(* PLC project TC3_TE1400_GeneratedModule_ModelBase2FM_FB, Beckhoff Automation GmbH & Co. KG TwinCAT 3 Function - TE1400 1.2.1228 *)
(* stored: companyURL www.beckhoff.com, creationDateTime 2017-03-29T12:16:05 *)

TYPE E_TcMatSimDataAreaType : (NotSpecified := 0, Standard, InputSrc, InputDst, OutputSrc, OutputDst, InternalDa, MArea, RetainDa);
END_TYPE

TYPE ST_TcMatSimObjectDataAreaInfo : STRUCT
  pPlcVar : PVOID;
  pModuleProcImg : PVOID;
  nSize : UDINT;
  nDataAreaId : UDINT;
  eDataAreaType : E_TcMatSimDataAreaType;
END_STRUCT;
END_TYPE

{attribute 'pack_mode' := '4'}
TYPE ST_ModelBase2FM_InitData : STRUCT
  Header : TComInitDataHdr;
  CallByHdr : TComInitDataElmHdr;
  CallBy : TctModuleCallByType;
  ExecutionSequenceHdr : TComInitDataElmHdr;
  ExecutionSequence : TctModuleExecutionSequenceType;
  StepSizeHdr : TComInitDataElmHdr;
  StepSize : TctStepSizeType;
  ExtendedFileAccessOIDHdr : TComInitDataElmHdr;
  ExtendedFileAccessOID : OTCID;
  ExtModeParametersHdr : TComInitDataElmHdr;
  ExtModeParameters : TctExtModeParametersType;
  ExecuteModelCodeHdr : TComInitDataElmHdr;
  ExecuteModelCode : BOOL;
  ModelParametersHdr : TComInitDataElmHdr;
  ModelParameters : P_model_base_2fm_T;
  ContextInfoArr_0_TaskOidHdr : TComInitDataElmHdr;
  ContextInfoArr_0_TaskOid : OTCID;
  ContextInfoArr_0_TaskPriorityHdr : TComInitDataElmHdr;
  ContextInfoArr_0_TaskPriority : UDINT;
  ContextInfoArr_0_TaskCycleTimeNsHdr : TComInitDataElmHdr;
  ContextInfoArr_0_TaskCycleTimeNs : UDINT;
  ContextInfoArr_0_TaskPortHdr : TComInitDataElmHdr;
  ContextInfoArr_0_TaskPort : UINT;
  ContextInfoArr_0_TaskSortOrderHdr : TComInitDataElmHdr;
  ContextInfoArr_0_TaskSortOrder : UDINT;
END_STRUCT;
END_TYPE

TYPE ST_ModelBase2FM_Input : STRUCT
  StatusWord_joint1 : UINT;
  MotorEncoder_joint1 : DINT;
  JointAbsEnc_joint1 : DINT;
  MotorCurrentAct_joint1 : INT;
  StatusWord_joint2 : UINT;
  MotorEncoder_joint2 : DINT;
  JointAbsEnc_joint2 : DINT;
  MotorCurrentAct_joint2 : INT;
  FTch1 : REAL;
  FTch2 : REAL;
  FTch3 : REAL;
  FTch4 : REAL;
  FTch5 : REAL;
  FTch6 : REAL;
  StatusWord_joint3 : UINT;
  MotorEncoder_joint3 : DINT;
  JointAbsEnc_joint3 : DINT;
  MotorCurrentAct_joint3 : INT;
  StatusWord_joint4 : UINT;
  MotorEncoder_joint4 : DINT;
  JointAbsEnc_joint4 : DINT;
  MotorCurrentAct_joint4 : INT;
  FTch7 : REAL;
  FTch8 : REAL;
  FTch9 : REAL;
  FTch10 : REAL;
  FTch11 : REAL;
  FTch12 : REAL;
END_STRUCT;
END_TYPE

TYPE ST_ModelBase2FM_Output : STRUCT
  EnableCircuit : BOOL;
  ControlWord_joint1 : UINT;
  ModesOfOperation_joint1 : SINT;
  TargetCurrent_joint1 : INT;
  ControlWord_joint2 : UINT;
  ModesOfOperation_joint2 : SINT;
  TargetCurrent_joint2 : INT;
  pause_logger : BOOL;
  EnableCircuit1 : BOOL;
  ControlWord_joint3 : UINT;
  ModesOfOperation_joint3 : SINT;
  TargetCurrent_joint3 : INT;
  ControlWord_joint4 : UINT;
  ModesOfOperation_joint4 : SINT;
  TargetCurrent_joint4 : INT;
END_STRUCT;
END_TYPE

FUNCTION_BLOCK FB_TcMatSimObject
  VAR_INPUT
    bWriteFbInputValues : BOOL := TRUE;  (* set this flag to write FB input values to the TcComObject's input DataAreas. This will overwrite the mapped input values before module execution. Set to FALSE to read the mapped input values from the TcComObject to the FB. *)
  END_VAR
  VAR
    pDataAreas : POINTER TO ST_TcMatSimObjectDataAreaInfo;  (* process image src and dst pointers and sizes *)
    nDataAreas : UDINT;
    ipObjSrv : ITComObjectServer;  (* global interface pointers *)
    ipTcComObj : ITComObject;  (* object interface pointers *)
    ipTcCyclic : ITcCyclic;
    ipTcPostCyclic : ITcPostCyclic;
    ipTcAdi : ITcADI;
    ipTask : ITcTask;  (* task interface pointers *)
    pInitData : POINTER TO TComInitDataHdr;  (* initial parameters *)
    hResult : HRESULT;  (* hResult of interface calls (0 if no error) *)
    moduleClsId : CLSID;  (* module class ID *)
    assignedClsId : CLSID;  (* expected/desired module class ID *)
    bClassIdVerified : BOOL;
    bDynInstance : BOOL;  (* flag indicating whether the module instance was created dynamically *)
    eInitialObjState : TCOM_STATE := TCOM_STATE.TCOM_STATE_INIT;  (* the object state at the time FB_init was called, FB_exit will try to switch to this state (only if this means to shift down) *)
  END_VAR

            
          

{attribute 'object_name' := 'ReleaseTcComInterface'}
METHOD ReleaseTcComInterface : HRESULT
  VAR
    nStateChangeCnt : DINT := 0;
  END_VAR
                  
IF (ipTcComObj<>0) THEN
  WHILE (State>eInitialObjState AND nStateChangeCnt<1000) DO
    State := eInitialObjState;
    nStateChangeCnt := nStateChangeCnt+1;
  END_WHILE
  ReleaseObjInterfaces();
  IF (bDynInstance) THEN
    ReleaseTcComInterface := TC3_MODULE.FW_ObjMgr_DeleteInstance(ADR(ipTcComObj));
  ELSE
    ipTcComObj.TcRelease();
  END_IF
  ipTcComObj := 0;
END_IF
                  
                
END_METHOD

{attribute 'object_name' := 'ReleaseObjInterfaces'}
METHOD ReleaseObjInterfaces : HRESULT
                  
// release interface pointers
IF (ipTcCyclic<>0) THEN
  ipTcCyclic.TcRelease();
  ipTcCyclic := 0;
END_IF
IF (ipTcPostCyclic<>0) THEN
  ipTcPostCyclic.TcRelease();
  ipTcPostCyclic := 0;
END_IF
IF (ipTcAdi<>0) THEN
  ipTcAdi.TcRelease();
  ipTcAdi := 0;
END_IF
                  
                
END_METHOD

{attribute 'object_name' := 'Internal_SetObjState'}
METHOD Internal_SetObjState
  VAR_INPUT
    hr : REFERENCE TO HRESULT;
    nextState : TCOM_STATE;
  END_VAR
                  
// verify class id
IF (SUCCEEDED(hr)) THEN
  hr := VerifyClassId();
END_IF

// switch object state
IF (SUCCEEDED(hr) AND nextState>=TCOM_STATE_INIT) THEN
  IF (ipTcComObj=0) THEN
    hr := Tc2_System.E_HRESULTAdsErr.NOINTERFACE;
  END_IF
  IF (ipObjSrv=0) THEN
    hr := Tc2_System.E_HRESULTAdsErr.NOINTERFACE;
  END_IF
  IF (SUCCEEDED(hr)) THEN
    hr := ipTcComObj.TcSetObjState(nextState,ipObjSrv,pInitData);
  END_IF
END_IF
                  
                
END_METHOD

{attribute 'object_name' := 'FB_init'}
METHOD FB_init : BOOL
  VAR_INPUT
    bInitRetains : BOOL;  (* init retain variables *)
    bInCopyCode : BOOL;  (* Online Change *)
    oid : OTCID;
  END_VAR
                  
FB_init := SUCCEEDED(Init(oid));
                  
                
END_METHOD

{attribute 'object_name' := 'GetObjPara'}
METHOD GetObjPara : HRESULT
  VAR_INPUT
    pid : PTCID;
    nData : UDINT;
    pData : PVOID;
  END_VAR
                  
IF (ipTcComObj=0) THEN
  GetObjPara := Tc2_System.E_HRESULTAdsErr.NOINTERFACE;
END_IF

IF (SUCCEEDED(GetObjPara)) THEN
  GetObjPara := ipTcComObj.TcGetObjPara(pid:=pid,nData,pData,0);
END_IF
                  
                
END_METHOD

{attribute 'object_name' := 'QueryObjInterface'}
METHOD QueryObjInterface
  VAR_INPUT
    hr : REFERENCE TO HRESULT;
    iid : REFERENCE TO IID;
    pipItf : POINTER TO ITcUnknown;
  END_VAR
  VAR CONSTANT
    pNull : PVOID := 0;
  END_VAR
                  
IF (SUCCEEDED(hr)) THEN
  IF (ipTcComObj=0) THEN
    hr := Tc2_System.E_HRESULTAdsErr.NOINTERFACE;
  ELSIF (pipItf^=ULINT_TO_DWORD(pNull)) THEN
    hr := ipTcComObj.TcQueryInterface(iid:= iid, pipItf:=pipItf);
  END_IF
END_IF
                  
                
END_METHOD

{attribute 'object_name' := 'SaveOnlineParametersForInit'}
METHOD SaveOnlineParametersForInit : HRESULT
  VAR
    idx : UINT;
    pInitElemHdr : POINTER TO TComInitDataElmHdr;
    pData : PVOID;
    nData : UDINT;
  END_VAR
  VAR CONSTANT
    nInitDataAlignment : UDINT := 4;
  END_VAR
                  IF (pInitData<>0) THEN
  pInitElemHdr := pInitData + SIZEOF(pInitData^);
  FOR idx:=1 TO pInitData^.uiElmCnt DO
    pData := pInitElemHdr + ULINT_TO_DWORD(SIZEOF(pInitElemHdr^));
    nData := pInitElemHdr^.cbData;
    SaveOnlineParametersForInit := GetObjPara(pInitElemHdr^.indexOffset,nData,pData);
    IF (FAILED(SaveOnlineParametersForInit)) THEN
      RETURN;
    END_IF
    pInitElemHdr := pData + (nInitDataAlignment*((nData + nInitDataAlignment - 1)/nInitDataAlignment));
  END_FOR
ELSE
	SaveOnlineParametersForInit := Tc2_System.E_HRESULTAdsErr.NOTINIT;
END_IF
                  
                
END_METHOD

{attribute 'object_name' := 'ResetHresult'}
METHOD ResetHresult
                  hResult := S_OK;
                
END_METHOD

{attribute 'object_name' := 'Execute'}
METHOD Execute : HRESULT
  VAR
    nDaIdx : UDINT;
    pCurDataArea : POINTER TO ST_TcMatSimObjectDataAreaInfo;
  END_VAR
                  
IF (SUCCEEDED(hResult)) THEN
  hResult := VerifyClassId();
END_IF

IF (SUCCEEDED(hResult) AND State<>TCOM_STATE_OP) THEN
  hResult := Tc2_System.E_HRESULTAdsErr.NOTREADY;
END_IF

// get image pointers
IF (SUCCEEDED(hResult)) THEN
  GetImagePtrs(hResult);
END_IF

// copy inputs
IF (pDataAreas<>0 AND bWriteFbInputValues) THEN
  FOR nDaIdx:=0 TO nDataAreas-1 DO
    IF (FAILED(hResult))THEN
      CONTINUE;
    END_IF
    pCurDataArea := pDataAreas + nDaIdx*SIZEOF(ST_TcMatSimObjectDataAreaInfo);
    IF ((pCurDataArea^.eDataAreaType <> E_TcMatSimDataAreaType.InputDst))THEN
      CONTINUE;
    END_IF
    IF (pCurDataArea^.pModuleProcImg<>0 AND pCurDataArea^.pPlcVar<>0) THEN
      MEMCPY(pCurDataArea^.pModuleProcImg,pCurDataArea^.pPlcVar,pCurDataArea^.nSize);
    ELSE
      hResult := Tc2_System.E_HRESULTAdsErr.NOINTERFACE;
    END_IF
  END_FOR
END_IF

// call cycle update
IF (SUCCEEDED(hResult)) THEN
  IF (ipTcCyclic<>0) THEN
    hResult := ipTcCyclic.CycleUpdate(ipTask:= ipTask, ipCaller:= 0, context:= 0);
  ELSE
    hResult := Tc2_System.E_HRESULTAdsErr.NOINTERFACE;
  END_IF
END_IF

// copy outputs
IF (pDataAreas<>0) THEN
  FOR nDaIdx:=0 TO nDataAreas-1 DO
    IF (FAILED(hResult))THEN
      CONTINUE;
    END_IF
    pCurDataArea := pDataAreas + nDaIdx*SIZEOF(ST_TcMatSimObjectDataAreaInfo);
    IF ((pCurDataArea^.eDataAreaType = E_TcMatSimDataAreaType.OutputSrc) OR NOT bWriteFbInputValues) THEN
      IF (pCurDataArea^.pModuleProcImg<>0 AND pCurDataArea^.pPlcVar<>0) THEN
        MEMCPY(pCurDataArea^.pPlcVar,pCurDataArea^.pModuleProcImg,pCurDataArea^.nSize);
      ELSE
        hResult := Tc2_System.E_HRESULTAdsErr.NOINTERFACE;
      END_IF
    END_IF
  END_FOR
END_IF


// call post cyclic update
IF (SUCCEEDED(hResult)) THEN
  IF (ipTcPostCyclic<>0) THEN
    hResult := ipTcPostCyclic.PostCyclicUpdate(ipTask:= 0, ipCaller:= 0, context:= 0);
  ELSE
    hResult := Tc2_System.E_HRESULTAdsErr.NOINTERFACE;
  END_IF
END_IF

ReleaseImagePtrs();

Execute := hResult;
                  
                
END_METHOD

{attribute 'object_name' := 'GetImagePtrs'}
METHOD GetImagePtrs
  VAR_INPUT
    hr : REFERENCE TO HRESULT;
  END_VAR
  VAR
    nDaIdx : UDINT;
    pCurDataArea : POINTER TO ST_TcMatSimObjectDataAreaInfo;
  END_VAR
                  
IF (ipTcAdi=0) THEN
  hr := Tc2_System.E_HRESULTAdsErr.NOINTERFACE;
END_IF
IF(State<>TCOM_STATE_OP)THEN
  hr := Tc2_System.E_HRESULTAdsErr.INVALIDSTATE;
END_IF


// get pointers to process images
IF (pDataAreas<>0) THEN
  FOR nDaIdx:=0 TO nDataAreas-1 DO
    pCurDataArea := pDataAreas + nDaIdx*SIZEOF(ST_TcMatSimObjectDataAreaInfo);
    IF (FAILED(hr))THEN
      CONTINUE;
    END_IF
    IF ((pCurDataArea^.eDataAreaType <> E_TcMatSimDataAreaType.InputDst) AND (pCurDataArea^.eDataAreaType <> E_TcMatSimDataAreaType.OutputSrc))THEN
      CONTINUE;
    END_IF
    IF (pCurDataArea^.pModuleProcImg=0 AND pCurDataArea^.nSize>0) THEN
      hr := ipTcAdi.GetImagePtr(size:= pCurDataArea^.nSize , offs:=0 , adi_x:=pCurDataArea^.nDataAreaId , ppData:=ADR(pCurDataArea^.pModuleProcImg));
    END_IF
  END_FOR
END_IF

IF (FAILED(hr)) THEN
  ReleaseImagePtrs();
END_IF
                  
                
END_METHOD

{attribute 'object_name' := 'VerifyClassId'}
METHOD VerifyClassId : HRESULT
  VAR
    emptyClsId : CLSID;
  END_VAR
                  memset(ADR(emptyClsId),0,SIZEOF(emptyClsId));
IF (bClassIdVerified) THEN
  // class ID was already verified
  VerifyClassId := Tc2_System.E_HRESULTAdsErr.HRESULT_ADS_NOERROR;
ELSIF (memcmp(ADR(assignedClsId),ADR(emptyClsId),SIZEOF(assignedClsId))=0) THEN
  // skip class ID verification if no assignedClsId specified
  VerifyClassId := Tc2_System.E_HRESULTAdsErr.HRESULT_ADS_NOERROR;
ELSE
  // verify class ID
  VerifyClassId := ReadModuleClassId();

  IF (SUCCEEDED(VerifyClassId)) THEN
    IF (memcmp(ADR(assignedClsId),ADR(moduleClsId),SIZEOF(assignedClsId))<>0) THEN
     VerifyClassId := Tc2_System.E_HRESULTAdsErr.INVALIDCLSID;
    END_IF
  END_IF
  bClassIdVerified := SUCCEEDED(VerifyClassId);
END_IF
                  
                
END_METHOD

{attribute 'object_name' := 'SetObjPara'}
METHOD SetObjPara : HRESULT
  VAR_INPUT
    pid : PTCID;
    nData : UDINT;
    pData : PVOID;
  END_VAR
                  
IF (ipTcComObj=0) THEN
  SetObjPara := Tc2_System.E_HRESULTAdsErr.NOINTERFACE;
END_IF

IF (SUCCEEDED(SetObjPara)) THEN
  SetObjPara := ipTcComObj.TcSetObjPara(pid:=pid,nData,pData,0);
END_IF
                  
                
END_METHOD

{attribute 'object_name' := 'QueryTcComInterface'}
METHOD QueryTcComInterface
  VAR_INPUT
    hr : REFERENCE TO HRESULT;
    oid : OTCID;
  END_VAR
                  
IF (ipObjSrv=0) THEN
  hr := Tc2_System.E_HRESULTAdsErr.NOINTERFACE;
END_IF

IF (SUCCEEDED(hr) AND ipTcComObj=0) THEN
  bDynInstance := FALSE;
  IF(oid>0) THEN
    // query interface of existing object
    hr := ipObjSrv.TcQueryObjectInterface(oid,IID_ITComObject,ADR(ipTcComObj));
  ELSE
    // create new instance and get the object interface
    hr := ipObjSrv.TcCreateInstance(assignedClsId,IID_ITComObject,ADR(ipTcComObj));
    IF (SUCCEEDED(hr)) THEN
      bDynInstance := TRUE;
      hr := ipTcComObj.TcSetObjectId(OTCID_CreateNewId);
    END_IF
  END_IF
  IF (SUCCEEDED(hr)) THEN
    eInitialObjState := State;
  END_IF
END_IF
                  
                
END_METHOD

{attribute 'object_name' := 'ReleaseImagePtrs'}
METHOD ReleaseImagePtrs : HRESULT
  VAR
    nDaIdx : UDINT;
    pCurDataArea : POINTER TO ST_TcMatSimObjectDataAreaInfo;
  END_VAR
                  
IF (ipTcAdi=0) THEN
  ReleaseImagePtrs := Tc2_System.E_HRESULTAdsErr.NOINTERFACE;
END_IF

IF (SUCCEEDED(ReleaseImagePtrs) AND pDataAreas<>0) THEN
  // release pointers to the simulink module process images
  FOR nDaIdx:=0 TO nDataAreas-1 DO
    pCurDataArea := pDataAreas + nDaIdx*SIZEOF(ST_TcMatSimObjectDataAreaInfo);

    IF (pCurDataArea^.pModuleProcImg<>0) THEN
      ipTcAdi.ReleaseImagePtr(pData:=pCurDataArea^.pModuleProcImg);
      pCurDataArea^.pModuleProcImg := 0;
    END_IF
  END_FOR
END_IF
                  
                
END_METHOD

{attribute 'object_name' := 'FB_exit'}
METHOD FB_exit : BOOL
  VAR_INPUT
    bInCopyCode : BOOL;  (* Online Change *)
  END_VAR
                  
IF (NOT bInCopyCode) THEN
  IF (ipObjSrv<>0) THEN
    ipObjSrv.TcRelease();
    ipObjSrv := 0;
  END_IF

  ReleaseTcComInterface();
END_IF
                  
                
END_METHOD

{attribute 'object_name' := 'InitObjName'}
METHOD InitObjName
  VAR_INPUT
    hr : REFERENCE TO HRESULT;
  END_VAR
  VAR
    objectName : STRING(255) := 'TempContr_PlcRtFbInstance';
    oid : OTCID;
  END_VAR
                  
IF (SUCCEEDED(hr)) THEN
  hr := ipTcComObj.TcGetObjectId(oid);
END_IF

IF (SUCCEEDED(hr) and bDynInstance) THEN
  objectName := TC2_STANDARD.CONCAT(objectName,'_');
  objectName := TC2_STANDARD.CONCAT(objectName,UDINT_TO_STRING(oid));
  hr := ipTcComObj.TcSetObjectName(ADR(objectName));
END_IF
                  
                
END_METHOD

{attribute 'object_name' := 'SetObjState'}
METHOD SetObjState : HRESULT
  VAR_INPUT
    finalState : TCOM_STATE;
  END_VAR
  VAR
    bShiftUp : BOOL;
    bShiftDown : BOOL;
    currentState : TCOM_STATE;
  END_VAR
                  
currentState := State;

bShiftUp := finalState>currentState;
bShiftDown := finalState<currentState;

// do not switch up on error
IF (FAILED(hresult)) THEN
  bShiftUp := FALSE;
END_IF
// reset existing error on switching down
IF (bShiftDown) THEN
  ResetHresult();
END_IF

// prepared state switch
CASE currentState OF
  TCOM_STATE_INIT:
    IF(bShiftUp) THEN
      QueryTcComInterface(hResult,0);
      Internal_SetObjState(hResult,TCOM_STATE.TCOM_STATE_PREOP);
      InitObjName(hResult);
    END_IF

  TCOM_STATE_PREOP:
    IF(bShiftUp) THEN
      Internal_SetObjState(hResult,TCOM_STATE.TCOM_STATE_SAFEOP);
      QueryObjInterfaces(hResult);
    ELSIF (bShiftDown) THEN
      Internal_SetObjState(hResult,TCOM_STATE.TCOM_STATE_INIT);
    END_IF

  TCOM_STATE_SAFEOP:
    IF(bShiftUp) THEN
      Internal_SetObjState(hResult,TCOM_STATE.TCOM_STATE_OP);
      QueryObjInterfaces(hResult);
    ELSIF (bShiftDown) THEN
      Internal_SetObjState(hResult,TCOM_STATE.TCOM_STATE_PREOP);
      ReleaseObjInterfaces();
    END_IF


  TCOM_STATE_OP:
    IF (bShiftDown) THEN
      Internal_SetObjState(hResult,TCOM_STATE.TCOM_STATE_SAFEOP);
    END_IF
END_CASE

SetObjState := hResult;
                  
                
END_METHOD

{attribute 'object_name' := 'QueryObjInterfaces'}
METHOD QueryObjInterfaces
  VAR_INPUT
    hr : REFERENCE TO HRESULT;
  END_VAR
                  
IF(State<TCOM_STATE_PREOP)THEN
  hr := Tc2_System.E_HRESULTAdsErr.INVALIDSTATE;
END_IF

//cyclic interface
QueryObjInterface(hr,IID_ITCCYCLIC,ADR(ipTcCyclic));
//post cyclic interface
QueryObjInterface(hr,IID_ITCPOSTCYCLIC,ADR(ipTcPostCyclic));
//adi interface
QueryObjInterface(hr,IID_ITcADI,ADR(ipTcAdi));
                  
                
END_METHOD

{attribute 'object_name' := 'Init'}
METHOD Init : HRESULT
  VAR_INPUT
    oid : OTCID;
  END_VAR
                  
// preinitialize variables
memset(ADR(moduleClsId),0,SIZEOF(moduleClsId));
bClassIdVerified := FALSE;
hResult := Tc2_System.E_HRESULTAdsErr.HRESULT_ADS_NOERROR;

// get object server
IF (ipObjSrv=0) THEN
  hResult := FW_ObjMgr_GetObjectServer(_AppInfo.ObjId,ADR(ipObjSrv));
END_IF

// try to get object interfaces
IF (SUCCEEDED(hresult)) THEN
  QueryTcComInterface(hResult,oid);
END_IF

// verify class id
IF (SUCCEEDED(hresult)) THEN
  hresult := VerifyClassId();
END_IF

// query interfaces, if the current state is higher than INIT
IF (SUCCEEDED(hresult) AND State>TCOM_STATE.TCOM_STATE_INIT) THEN
  QueryObjInterfaces(hResult);
END_IF

// return value
Init := hresult;
                  
                
END_METHOD

{attribute 'object_name' := 'ReadModuleClassId'}
METHOD ReadModuleClassId : HRESULT
  VAR
    emptyClsId : CLSID;
  END_VAR
                  memset(ADR(emptyClsId),0,SIZEOF(emptyClsId));
IF (memcmp(ADR(moduleClsId),ADR(emptyClsId),SIZEOF(moduleClsId))=0) THEN
  IF (ipTcComObj=0) THEN
    ReadModuleClassId := Tc2_System.E_HRESULTAdsErr.NOINTERFACE;
  END_IF

  //objectClsId := clsid;
  IF (SUCCEEDED(ReadModuleClassId)) THEN
    ReadModuleClassId := ipTcComObj.GetClassId(moduleClsId);
  END_IF
END_IF
                
END_METHOD

METHOD PUBLIC AssignClassId
VAR_INPUT
	clsId : CLSID;
END_VAR
                  assignedClsId := clsId;
bClassIdVerified := false;
                  
                
END_METHOD

PROPERTY Error : BOOL
GET
                    Error := FAILED(hResult);
                  
END_GET
END_PROPERTY

METHOD PUBLIC SetDataAreaInfo
VAR_INPUT
  pDataAreas: POINTER TO ST_TcMatSimObjectDataAreaInfo;
  nDataAreas: UDINT;
END_VAR
                  
THIS^.nDataAreas := nDataAreas;
THIS^.pDataAreas := pDataAreas;
                  
                
END_METHOD

METHOD PUBLIC SetInitDataInfo
VAR_INPUT
  pInitData : POINTER TO TComInitDataHdr;
END_VAR
                  this^.pInitData := pInitData;
                
END_METHOD

PROPERTY ClassId : CLSID
GET
                    hResult := ReadModuleClassId();
ClassId := moduleClsId;
                    
                  
END_GET
END_PROPERTY

PROPERTY State : TCOM_STATE
GET
  VAR
    hr : HRESULT := S_OK;
    eObjState : TCOM_STATE;
  END_VAR
                    
IF (ipTcComObj<>0) THEN
  hr := ipTcComObj.TcGetObjState(ADR(eObjState));
IF (FAILED(hr)) THEN
  eObjState := TCOM_STATE.TCOM_STATE_INIT;
END_IF
ELSE
  eObjState := TCOM_STATE.TCOM_STATE_INIT;
END_IF
State := eObjState;
                    
                  
END_GET
SET
                    SetObjState(State);
                  
END_SET
END_PROPERTY

PROPERTY ErrorCode : HRESULT
GET
                    ErrorCode := hResult;
                  
END_GET
END_PROPERTY
END_FUNCTION_BLOCK

{attribute 'TcDependOnClassFactory' := 'ModelBase2FM'}
FUNCTION_BLOCK FB_ModelBase2FM EXTENDS FB_TcMatSimObject
  VAR_INPUT
    stInput : ST_ModelBase2FM_Input;
  END_VAR
  VAR_OUTPUT
    stOutput : ST_ModelBase2FM_Output;
  END_VAR
  VAR
    stInitData : ST_ModelBase2FM_InitData;
    arrDataAreas : ARRAY[1..2] OF ST_TcMatSimObjectDataAreaInfo;
    bParametersVerified : BOOL;
  END_VAR

            
          

{attribute 'object_name' := 'Internal_SetObjState'}
METHOD Internal_SetObjState
  VAR_INPUT
    hr : REFERENCE TO HRESULT;
    nextState : TCOM_STATE;
  END_VAR
                  
// update pointer to InitData structure
SetInitDataInfo(ADR(stInitData));
// call base method
SUPER^.Internal_SetObjState(hr,nextState);
                  
                
END_METHOD

{attribute 'object_name' := 'SaveOnlineParametersForInit'}
METHOD SaveOnlineParametersForInit : HRESULT
  VAR
    idx : UINT;
    pInitElemHdr : POINTER TO TComInitDataElmHdr;
    pData : PVOID;
    nData : UDINT;
  END_VAR
  VAR CONSTANT
    nInitDataAlignment : UDINT := 4;
  END_VAR
                  
// update pointer to InitData structure
SetInitDataInfo(ADR(stInitData));
// call base method
SaveOnlineParametersForInit := SUPER^.SaveOnlineParametersForInit();
                  
                
END_METHOD

METHOD FB_init : BOOL
  VAR_INPUT
    bInitRetains : BOOL;  (* if TRUE, the retain variables are initialized (warm start / cold start) *)
    bInCopyCode : BOOL;  (* if TRUE, the instance afterwards gets moved into the copy code (online change) *)
    oid : OTCID;
  END_VAR
  VAR
    clsId : CLSID;
  END_VAR
                  
// initialize flags
bParametersVerified := false;
                    
// set module class id for compatibility check
clsId.Data1 := 16#36160af7;
clsId.Data2 := 16#e4ae;
clsId.Data3 := 16#44ca;
clsId.Data4[0] := 16#81;
clsId.Data4[1] := 16#8b;
clsId.Data4[2] := 16#1e;
clsId.Data4[3] := 16#af;
clsId.Data4[4] := 16#06;
clsId.Data4[5] := 16#99;
clsId.Data4[6] := 16#96;
clsId.Data4[7] := 16#6e;

AssignClassId(clsId);
                    
// initialize InitData structure with default values              
stInitData.CallByHdr.indexGroup := 0;
stInitData.CallByHdr.indexOffset := 16#00000000;
stInitData.CallByHdr.cbData := SIZEOF(stInitData.CallBy);
stInitData.CallBy := TctModuleCallByType.CyclicTask;
stInitData.ExecutionSequenceHdr.indexGroup := 0;
stInitData.ExecutionSequenceHdr.indexOffset := 16#00000001;
stInitData.ExecutionSequenceHdr.cbData := SIZEOF(stInitData.ExecutionSequence);
stInitData.ExecutionSequence := TctModuleExecutionSequenceType.StateUpdateAfterOutputMapping;
stInitData.StepSizeHdr.indexGroup := 0;
stInitData.StepSizeHdr.indexOffset := 16#00000002;
stInitData.StepSizeHdr.cbData := SIZEOF(stInitData.StepSize);
stInitData.StepSize := TctStepSizeType.RequireMatchingTaskCycleTime;
stInitData.ExtendedFileAccessOIDHdr.indexGroup := 0;
stInitData.ExtendedFileAccessOIDHdr.indexOffset := 16#00000005;
stInitData.ExtendedFileAccessOIDHdr.cbData := SIZEOF(stInitData.ExtendedFileAccessOID);
stInitData.ExtendedFileAccessOID := 0;
stInitData.ExtModeParametersHdr.indexGroup := 0;
stInitData.ExtModeParametersHdr.indexOffset := 16#bf002000;
stInitData.ExtModeParametersHdr.cbData := SIZEOF(stInitData.ExtModeParameters);
stInitData.ExtModeParameters.ConnectionTimeout := 3;
stInitData.ExtModeParameters.InitIncomingPktBufferSize := 10000;
stInitData.ExtModeParameters.InitOutgoingPktBufferSize := 10000;
stInitData.ExtModeParameters.Activated := 1;
stInitData.ExtModeParameters.AllowExecutionCommands := 1;
stInitData.ExtModeParameters.WaitForStartCommand := 0;
stInitData.ExtModeParameters.AllowParameterChange := 1;
stInitData.ExecuteModelCodeHdr.indexGroup := 0;
stInitData.ExecuteModelCodeHdr.indexOffset := 16#00000008;
stInitData.ExecuteModelCodeHdr.cbData := SIZEOF(stInitData.ExecuteModelCode);
stInitData.ExecuteModelCode := 1;
stInitData.ModelParametersHdr.indexGroup := 0;
stInitData.ModelParametersHdr.indexOffset := 16#83000000;
stInitData.ModelParametersHdr.cbData := SIZEOF(stInitData.ModelParameters);
stInitData.ModelParameters.FM1.HomeLocationOpSpace[0] := 0;
stInitData.ModelParameters.FM1.HomeLocationOpSpace[1] := 0.25;
stInitData.ModelParameters.FM1.HomeLocationSize := 0.01;
stInitData.ModelParameters.FM1.DynModParams[0] := 0.001597109;
stInitData.ModelParameters.FM1.DynModParams[1] := 0.001580786;
stInitData.ModelParameters.FM1.DynModParams[2] := 0.0702826;
stInitData.ModelParameters.FM1.DynModParams[3] := 0.07988736;
stInitData.ModelParameters.FM1.DynModParams[4] := -0;
stInitData.ModelParameters.FM1.DynModParams[5] := 0.1006366;
stInitData.ModelParameters.FM1.DynModParams[6] := -0;
stInitData.ModelParameters.FM1.Actuator1.JointAbsoluteEncoderCounts_rev := 65536;
stInitData.ModelParameters.FM1.Actuator1.AbsEncoderOffset := 5.303223547422882;
stInitData.ModelParameters.FM1.Actuator1.MotorEncoderCounts_rev := 4096;
stInitData.ModelParameters.FM1.Actuator1.FOAWNoiseLevel := 0.0003834951969714103;
stInitData.ModelParameters.FM1.Actuator1.transmissionRatio := 7.2976;
stInitData.ModelParameters.FM1.Actuator1.motorTorqueConstant := 0.08486;
stInitData.ModelParameters.FM1.Actuator1.drivePeakCurrent := 20;
stInitData.ModelParameters.FM1.Actuator1.AbsoluteMaximumTorque_Nm := 8;
stInitData.ModelParameters.FM1.Actuator1.TransmissionSlipAngleGuardMax := 0.08726646259971647;
stInitData.ModelParameters.FM1.Actuator1.JointPositionGuardMin := -0.4363323129985824;
stInitData.ModelParameters.FM1.Actuator1.JointPositionGuardMax := 2.356194490192345;
stInitData.ModelParameters.FM1.Actuator2.JointAbsoluteEncoderCounts_rev := 65536;
stInitData.ModelParameters.FM1.Actuator2.AbsEncoderOffset := 7.340133727728301;
stInitData.ModelParameters.FM1.Actuator2.MotorEncoderCounts_rev := 4096;
stInitData.ModelParameters.FM1.Actuator2.FOAWNoiseLevel := 0.0003834951969714103;
stInitData.ModelParameters.FM1.Actuator2.transmissionRatio := 7.331;
stInitData.ModelParameters.FM1.Actuator2.motorTorqueConstant := 0.08486;
stInitData.ModelParameters.FM1.Actuator2.drivePeakCurrent := 20;
stInitData.ModelParameters.FM1.Actuator2.AbsoluteMaximumTorque_Nm := 8;
stInitData.ModelParameters.FM1.Actuator2.TransmissionSlipAngleGuardMax := 0.08726646259971647;
stInitData.ModelParameters.FM1.Actuator2.JointPositionGuardMin := 0.7853981633974483;
stInitData.ModelParameters.FM1.Actuator2.JointPositionGuardMax := 3.577924966588375;
stInitData.ModelParameters.FM1.FTSensor.MaxAllowableForcesTorqueSensor[0] := 70;
stInitData.ModelParameters.FM1.FTSensor.MaxAllowableForcesTorqueSensor[1] := 70;
stInitData.ModelParameters.FM1.FTSensor.MaxAllowableForcesTorqueSensor[2] := 140;
stInitData.ModelParameters.FM1.FTSensor.MaxAllowableForcesTorqueSensor[3] := 1.4;
stInitData.ModelParameters.FM1.FTSensor.MaxAllowableForcesTorqueSensor[4] := 1.4;
stInitData.ModelParameters.FM1.FTSensor.MaxAllowableForcesTorqueSensor[5] := 1.4;
stInitData.ModelParameters.FM1.FTSensor.TransformationMatrixSide := 1;
stInitData.ModelParameters.FM2.HomeLocationOpSpace[0] := 0;
stInitData.ModelParameters.FM2.HomeLocationOpSpace[1] := 0.25;
stInitData.ModelParameters.FM2.HomeLocationSize := 0.01;
stInitData.ModelParameters.FM2.DynModParams[0] := 0.001597109;
stInitData.ModelParameters.FM2.DynModParams[1] := 0.001580786;
stInitData.ModelParameters.FM2.DynModParams[2] := 0.0702826;
stInitData.ModelParameters.FM2.DynModParams[3] := 0.07988736;
stInitData.ModelParameters.FM2.DynModParams[4] := -0;
stInitData.ModelParameters.FM2.DynModParams[5] := 0.1006366;
stInitData.ModelParameters.FM2.DynModParams[6] := -0;
stInitData.ModelParameters.FM2.Actuator1.JointAbsoluteEncoderCounts_rev := 65536;
stInitData.ModelParameters.FM2.Actuator1.AbsEncoderOffset := 3.23580094055001;
stInitData.ModelParameters.FM2.Actuator1.MotorEncoderCounts_rev := 4096;
stInitData.ModelParameters.FM2.Actuator1.FOAWNoiseLevel := 0.0003834951969714103;
stInitData.ModelParameters.FM2.Actuator1.transmissionRatio := 7.3607;
stInitData.ModelParameters.FM2.Actuator1.motorTorqueConstant := 0.08486;
stInitData.ModelParameters.FM2.Actuator1.drivePeakCurrent := 20;
stInitData.ModelParameters.FM2.Actuator1.AbsoluteMaximumTorque_Nm := 8;
stInitData.ModelParameters.FM2.Actuator1.TransmissionSlipAngleGuardMax := 0.08726646259971647;
stInitData.ModelParameters.FM2.Actuator1.JointPositionGuardMin := -0.4363323129985824;
stInitData.ModelParameters.FM2.Actuator1.JointPositionGuardMax := 2.356194490192345;
stInitData.ModelParameters.FM2.Actuator2.JointAbsoluteEncoderCounts_rev := 65536;
stInitData.ModelParameters.FM2.Actuator2.AbsEncoderOffset := 4.445224359590367;
stInitData.ModelParameters.FM2.Actuator2.MotorEncoderCounts_rev := 4096;
stInitData.ModelParameters.FM2.Actuator2.FOAWNoiseLevel := 0.0003834951969714103;
stInitData.ModelParameters.FM2.Actuator2.transmissionRatio := 7.32214;
stInitData.ModelParameters.FM2.Actuator2.motorTorqueConstant := 0.08486;
stInitData.ModelParameters.FM2.Actuator2.drivePeakCurrent := 20;
stInitData.ModelParameters.FM2.Actuator2.AbsoluteMaximumTorque_Nm := 8;
stInitData.ModelParameters.FM2.Actuator2.TransmissionSlipAngleGuardMax := 0.08726646259971647;
stInitData.ModelParameters.FM2.Actuator2.JointPositionGuardMin := 0.7853981633974483;
stInitData.ModelParameters.FM2.Actuator2.JointPositionGuardMax := 3.577924966588375;
stInitData.ModelParameters.FM2.FTSensor.MaxAllowableForcesTorqueSensor[0] := 70;
stInitData.ModelParameters.FM2.FTSensor.MaxAllowableForcesTorqueSensor[1] := 70;
stInitData.ModelParameters.FM2.FTSensor.MaxAllowableForcesTorqueSensor[2] := 140;
stInitData.ModelParameters.FM2.FTSensor.MaxAllowableForcesTorqueSensor[3] := 1.4;
stInitData.ModelParameters.FM2.FTSensor.MaxAllowableForcesTorqueSensor[4] := 1.4;
stInitData.ModelParameters.FM2.FTSensor.MaxAllowableForcesTorqueSensor[5] := 1.4;
stInitData.ModelParameters.FM2.FTSensor.TransformationMatrixSide := 1;
stInitData.ModelParameters.Lb := 0.07000000000000001;
stInitData.ModelParameters.Lf := 0.238;
stInitData.ModelParameters.Lu := 0.153;
stInitData.ModelParameters.sampleTime := 0.001;
stInitData.ModelParameters.DiscreteDerivative_ICPrevScaled := 0;
stInitData.ModelParameters.DiscreteDerivative_ICPrevScal_b := 0;
stInitData.ModelParameters.DiscreteDerivative_ICPrevScal_a := 0;
stInitData.ModelParameters.DiscreteDerivative_ICPrevScal_h := 0;
stInitData.ModelParameters.DiscreteDerivative_ICPrevScal_j := 0;
stInitData.ModelParameters.DiscreteDerivative_ICPrevScal_k := 0;
stInitData.ModelParameters.DiscreteDerivative_ICPrevScal_i := 0;
stInitData.ModelParameters.DiscreteDerivative_ICPrevScal_o := 0;
stInitData.ModelParameters.CompareToConstant_const := 201;
stInitData.ModelParameters.CompareToConstant_const_b := 0;
stInitData.ModelParameters.CompareToConstant_const_a := 201;
stInitData.ModelParameters.CompareToConstant_const_e := 0;
stInitData.ModelParameters.CompareToConstant_const_aw := 4;
stInitData.ModelParameters.CompareToConstant_const_c := 4;
stInitData.ModelParameters.CompareToConstant1_const := 2.75;
stInitData.ModelParameters.CompareToConstant_const_d := 4;
stInitData.ModelParameters.CompareToConstant_const_m := 4;
stInitData.ModelParameters.CompareToConstant1_const_m := 2.75;
stInitData.ModelParameters.DetectChange_vinit := 0;
stInitData.ModelParameters.DetectChange_vinit_h := 0;
stInitData.ModelParameters.DetectChange_vinit_g := 0;
stInitData.ModelParameters.DetectChange_vinit_b := 0;
stInitData.ModelParameters.ErrorHasOccurred_initial_condit := 0;
stInitData.ModelParameters.ErrorHasOccurred_initial_cond_a := 0;
stInitData.ModelParameters.ErrorHasOccurred_initial_cond_f := 0;
stInitData.ModelParameters.ErrorHasOccurred_initial_cond_k := 0;
stInitData.ModelParameters.DetectRisePositive_vinit := 0;
stInitData.ModelParameters.DetectRisePositive1_vinit := 0;
stInitData.ModelParameters.DetectRisePositive_vinit_c := 0;
stInitData.ModelParameters.DetectRisePositive1_vinit_i := 0;
stInitData.ModelParameters.DetectRisePositive_vinit_m := 0;
stInitData.ModelParameters.DetectRisePositive1_vinit_b := 0;
stInitData.ModelParameters.DetectRisePositive_vinit_n := 0;
stInitData.ModelParameters.DetectRisePositive1_vinit_j := 0;
stInitData.ModelParameters.DetectIncrease_vinit := 0;
stInitData.ModelParameters.DetectIncrease_vinit_f := 0;
stInitData.ModelParameters.JointTorqueDes_Nm_Y0[0] := 0;
stInitData.ModelParameters.JointTorqueDes_Nm_Y0[1] := 0;
stInitData.ModelParameters.Constant3_Value[0] := 0;
stInitData.ModelParameters.Constant3_Value[1] := 0;
stInitData.ModelParameters.JointTorqueDes_Nm_Y0_p[0] := 0;
stInitData.ModelParameters.JointTorqueDes_Nm_Y0_p[1] := 0;
stInitData.ModelParameters.Constant3_Value_h[0] := 0;
stInitData.ModelParameters.Constant3_Value_h[1] := 0;
stInitData.ModelParameters.JointTorqueDes_Nm_Y0_i[0] := 0;
stInitData.ModelParameters.JointTorqueDes_Nm_Y0_i[1] := 0;
stInitData.ModelParameters.Constant3_Value_h5[0] := 0;
stInitData.ModelParameters.Constant3_Value_h5[1] := 0;
stInitData.ModelParameters.JointTorqueDes_Nm_Y0_m[0] := 0;
stInitData.ModelParameters.JointTorqueDes_Nm_Y0_m[1] := 0;
stInitData.ModelParameters.Constant3_Value_b[0] := 0;
stInitData.ModelParameters.Constant3_Value_b[1] := 0;
stInitData.ModelParameters.EnableDrives_Value := 0;
stInitData.ModelParameters.Constant_Value := 0;
stInitData.ModelParameters.UseActuator_Value := 1;
stInitData.ModelParameters.CalibrateManually_Value := 0;
stInitData.ModelParameters.Memory_X0 := 0;
stInitData.ModelParameters.FreqHz_Value := 20;
stInitData.ModelParameters.UnitDelay_InitialCondition := 0;
stInitData.ModelParameters.TSamp_WtEt := 1000;
stInitData.ModelParameters.FreqHz_Value_e := 100;
stInitData.ModelParameters.UnitDelay_InitialCondition_e := 0;
stInitData.ModelParameters.Constant_Value_m := 6.283185307179586;
stInitData.ModelParameters.AbsoluteMaximumTorque_Nm_Value := 8;
stInitData.ModelParameters.Bias_Bias := 0.5;
stInitData.ModelParameters.InhibitTime_s_Value := 2;
stInitData.ModelParameters.Memory1_1_X0 := 0;
stInitData.ModelParameters.DisableDrives_Value := 0;
stInitData.ModelParameters.Constant_Value_f := 0;
stInitData.ModelParameters.PreventAlgebraicLoop_X0 := 0;
stInitData.ModelParameters.PreventAlgebraicLoop_X0_a := 0;
stInitData.ModelParameters.Constant_Value_fn := 0;
stInitData.ModelParameters.AvoidAlgebraicLoop_X0 := 0;
stInitData.ModelParameters.Constant_Value_i := 0;
stInitData.ModelParameters.UseActuator_Value_g := 1;
stInitData.ModelParameters.CalibrateManually_Value_p := 0;
stInitData.ModelParameters.FreqHz_Value_j := 20;
stInitData.ModelParameters.UnitDelay_InitialCondition_f := 0;
stInitData.ModelParameters.TSamp_WtEt_o := 1000;
stInitData.ModelParameters.FreqHz_Value_c := 100;
stInitData.ModelParameters.UnitDelay_InitialCondition_c := 0;
stInitData.ModelParameters.Constant_Value_iv := 6.283185307179586;
stInitData.ModelParameters.AbsoluteMaximumTorque_Nm_Valu_n := 8;
stInitData.ModelParameters.Bias_Bias_c := 0.5;
stInitData.ModelParameters.InhibitTime_s_Value_b := 2;
stInitData.ModelParameters.Memory1_1_X0_i := 0;
stInitData.ModelParameters.Constant_Value_o := 0;
stInitData.ModelParameters.Constant_Value_ok := 0;
stInitData.ModelParameters.TimePerState_ms_Value[0] := 50;
stInitData.ModelParameters.TimePerState_ms_Value[1] := 50;
stInitData.ModelParameters.TimePerState_ms_Value[2] := 150;
stInitData.ModelParameters.TimePerState_ms_Value[3] := 150;
stInitData.ModelParameters.SetModeOp_val_slx_Value := 10;
stInitData.ModelParameters.Requestedstate_Value := 0;
stInitData.ModelParameters.AvoidAlgebraicLoop_X0_a := 0;
stInitData.ModelParameters.Gain_Gain := 1;
stInitData.ModelParameters.Gain_Gain_e := 1;
stInitData.ModelParameters.Constant2_Value := 0.05;
stInitData.ModelParameters.CalibrateManually_Value_j := 0;
stInitData.ModelParameters.Memory_X0_e := 0;
stInitData.ModelParameters.FreqHz_Value_f := 20;
stInitData.ModelParameters.UnitDelay_InitialCondition_ed := 0;
stInitData.ModelParameters.CalibrateManually_Value_g := 0;
stInitData.ModelParameters.FreqHz_Value_cf := 20;
stInitData.ModelParameters.UnitDelay_InitialCondition_er := 0;
stInitData.ModelParameters.Gain_Gain_b := 1;
stInitData.ModelParameters.Gain_Gain_ev := 1;
stInitData.ModelParameters.Constant1_Value[0] := 0;
stInitData.ModelParameters.Constant1_Value[1] := 0;
stInitData.ModelParameters.Merge1_InitialOutput[0] := 0;
stInitData.ModelParameters.Merge1_InitialOutput[1] := 0;
stInitData.ModelParameters.Kp_Gain := 0;
stInitData.ModelParameters.Merge2_InitialOutput[0] := 0;
stInitData.ModelParameters.Merge2_InitialOutput[1] := 0;
stInitData.ModelParameters.Kd_Gain := 0;
stInitData.ModelParameters.Kp1_Gain := 100;
stInitData.ModelParameters.Gain_Gain_m := 1.5;
stInitData.ModelParameters.Gain_Gain_l := 1.5;
stInitData.ModelParameters.Kd1_Gain := 2;
stInitData.ModelParameters.Gain_Gain_d := 0;
stInitData.ModelParameters.Saturation_UpperSat := 4;
stInitData.ModelParameters.Saturation_LowerSat := -4;
stInitData.ModelParameters.TimePerState_ms_Value_d[0] := 50;
stInitData.ModelParameters.TimePerState_ms_Value_d[1] := 50;
stInitData.ModelParameters.TimePerState_ms_Value_d[2] := 150;
stInitData.ModelParameters.TimePerState_ms_Value_d[3] := 150;
stInitData.ModelParameters.SetModeOp_val_slx_Value_n := 10;
stInitData.ModelParameters.Constant_Value_a := 0;
stInitData.ModelParameters.UseActuator_Value_a := 1;
stInitData.ModelParameters.TSamp_WtEt_l := 1000;
stInitData.ModelParameters.FreqHz_Value_a := 100;
stInitData.ModelParameters.UnitDelay_InitialCondition_fl := 0;
stInitData.ModelParameters.Constant_Value_d := 6.283185307179586;
stInitData.ModelParameters.AbsoluteMaximumTorque_Nm_Valu_l := 8;
stInitData.ModelParameters.Bias_Bias_p := 0.5;
stInitData.ModelParameters.InhibitTime_s_Value_m := 2;
stInitData.ModelParameters.Memory1_1_X0_h := 0;
stInitData.ModelParameters.Constant_Value_b := 0;
stInitData.ModelParameters.PreventAlgebraicLoop_X0_d := 0;
stInitData.ModelParameters.PreventAlgebraicLoop_X0_g := 0;
stInitData.ModelParameters.Constant_Value_iq := 0;
stInitData.ModelParameters.AvoidAlgebraicLoop_X0_l := 0;
stInitData.ModelParameters.Constant_Value_f0 := 0;
stInitData.ModelParameters.UseActuator_Value_d := 1;
stInitData.ModelParameters.TSamp_WtEt_ll := 1000;
stInitData.ModelParameters.FreqHz_Value_b := 100;
stInitData.ModelParameters.UnitDelay_InitialCondition_i := 0;
stInitData.ModelParameters.Constant_Value_a1 := 6.283185307179586;
stInitData.ModelParameters.AbsoluteMaximumTorque_Nm_Valu_e := 8;
stInitData.ModelParameters.Bias_Bias_o := 0.5;
stInitData.ModelParameters.InhibitTime_s_Value_j := 2;
stInitData.ModelParameters.Memory1_1_X0_a := 0;
stInitData.ModelParameters.Constant_Value_i3 := 0;
stInitData.ModelParameters.Constant_Value_g := 0;
stInitData.ModelParameters.TimePerState_ms_Value_k[0] := 50;
stInitData.ModelParameters.TimePerState_ms_Value_k[1] := 50;
stInitData.ModelParameters.TimePerState_ms_Value_k[2] := 150;
stInitData.ModelParameters.TimePerState_ms_Value_k[3] := 150;
stInitData.ModelParameters.SetModeOp_val_slx_Value_i := 10;
stInitData.ModelParameters.AvoidAlgebraicLoop_X0_m := 0;
stInitData.ModelParameters.Constant2_Value_f := 0.05;
stInitData.ModelParameters.Merge1_InitialOutput_i[0] := 0;
stInitData.ModelParameters.Merge1_InitialOutput_i[1] := 0;
stInitData.ModelParameters.Kp_Gain_m := 0;
stInitData.ModelParameters.Merge2_InitialOutput_m[0] := 0;
stInitData.ModelParameters.Merge2_InitialOutput_m[1] := 0;
stInitData.ModelParameters.Kd_Gain_l := 0;
stInitData.ModelParameters.Kp1_Gain_g := 100;
stInitData.ModelParameters.Gain_Gain_h := 1.5;
stInitData.ModelParameters.Gain_Gain_g := 1.5;
stInitData.ModelParameters.Kd1_Gain_d := 2;
stInitData.ModelParameters.Gain_Gain_p := 0;
stInitData.ModelParameters.Saturation_UpperSat_j := 4;
stInitData.ModelParameters.Saturation_LowerSat_j := -4;
stInitData.ModelParameters.TimePerState_ms_Value_c[0] := 50;
stInitData.ModelParameters.TimePerState_ms_Value_c[1] := 50;
stInitData.ModelParameters.TimePerState_ms_Value_c[2] := 150;
stInitData.ModelParameters.TimePerState_ms_Value_c[3] := 150;
stInitData.ModelParameters.SetModeOp_val_slx_Value_p := 10;
stInitData.ModelParameters.TSamp_WtEt_n := 1000;
stInitData.ModelParameters.FreqHz_Value_o := 150;
stInitData.ModelParameters.UnitDelay_InitialCondition_k := 0;
stInitData.ModelParameters.TSamp_WtEt_f := 1000;
stInitData.ModelParameters.FreqHz_Value_k := 150;
stInitData.ModelParameters.UnitDelay_InitialCondition_d := 0;
stInitData.ModelParameters.TSamp_WtEt_h := 1000;
stInitData.ModelParameters.FreqHz_Value_i := 150;
stInitData.ModelParameters.UnitDelay_InitialCondition_j := 0;
stInitData.ModelParameters.TSamp_WtEt_c := 1000;
stInitData.ModelParameters.FreqHz_Value_bi := 150;
stInitData.ModelParameters.UnitDelay_InitialCondition_o := 0;
stInitData.ModelParameters.Merge3_InitialOutput[0] := 0;
stInitData.ModelParameters.Merge3_InitialOutput[1] := 0;
stInitData.ModelParameters.Memory1_10_X0 := 0;
stInitData.ModelParameters.Memory1_11_X0 := 0;
stInitData.ModelParameters.Memory1_2_X0 := 0;
stInitData.ModelParameters.Memory1_3_X0 := 0;
stInitData.ModelParameters.Memory1_4_X0 := 0;
stInitData.ModelParameters.Memory1_5_X0 := 0;
stInitData.ModelParameters.Memory1_6_X0 := 0;
stInitData.ModelParameters.Memory1_7_X0 := 0;
stInitData.ModelParameters.Memory1_8_X0 := 0;
stInitData.ModelParameters.Memory1_9_X0 := 0;
stInitData.ModelParameters.Memory1_10_X0_i := 0;
stInitData.ModelParameters.Memory1_11_X0_i := 0;
stInitData.ModelParameters.Memory1_2_X0_i := 0;
stInitData.ModelParameters.Memory1_3_X0_i := 0;
stInitData.ModelParameters.Memory1_4_X0_i := 0;
stInitData.ModelParameters.Memory1_5_X0_i := 0;
stInitData.ModelParameters.Memory1_6_X0_i := 0;
stInitData.ModelParameters.Memory1_7_X0_i := 0;
stInitData.ModelParameters.Memory1_8_X0_i := 0;
stInitData.ModelParameters.Memory1_9_X0_i := 0;
stInitData.ModelParameters.Merge3_InitialOutput_j[0] := 0;
stInitData.ModelParameters.Merge3_InitialOutput_j[1] := 0;
stInitData.ModelParameters.Memory1_10_X0_h := 0;
stInitData.ModelParameters.Memory1_11_X0_h := 0;
stInitData.ModelParameters.Memory1_2_X0_h := 0;
stInitData.ModelParameters.Memory1_3_X0_h := 0;
stInitData.ModelParameters.Memory1_4_X0_h := 0;
stInitData.ModelParameters.Memory1_5_X0_h := 0;
stInitData.ModelParameters.Memory1_6_X0_h := 0;
stInitData.ModelParameters.Memory1_7_X0_h := 0;
stInitData.ModelParameters.Memory1_8_X0_h := 0;
stInitData.ModelParameters.Memory1_9_X0_h := 0;
stInitData.ModelParameters.Memory1_10_X0_a := 0;
stInitData.ModelParameters.Memory1_11_X0_a := 0;
stInitData.ModelParameters.Memory1_2_X0_a := 0;
stInitData.ModelParameters.Memory1_3_X0_a := 0;
stInitData.ModelParameters.Memory1_4_X0_a := 0;
stInitData.ModelParameters.Memory1_5_X0_a := 0;
stInitData.ModelParameters.Memory1_6_X0_a := 0;
stInitData.ModelParameters.Memory1_7_X0_a := 0;
stInitData.ModelParameters.Memory1_8_X0_a := 0;
stInitData.ModelParameters.Memory1_9_X0_a := 0;
stInitData.ModelParameters.Recorddata1yes0no_Value := 0;
stInitData.ModelParameters.Gain_Gain_f := 1;
stInitData.ModelParameters.ManualSwitch_CurrentSetting := 0;
stInitData.ModelParameters.ManualSwitch_CurrentSetting_f := 0;
stInitData.ModelParameters.ManualSwitch_CurrentSetting_j := 0;
stInitData.ModelParameters.ManualSwitch_CurrentSetting_n := 0;
stInitData.ModelParameters.Memory1_X0 := 0;
stInitData.ModelParameters.Memory_X0_f := 0;
stInitData.ModelParameters.Logic_table[0] := 0;
stInitData.ModelParameters.Logic_table[1] := 1;
stInitData.ModelParameters.Logic_table[2] := 0;
stInitData.ModelParameters.Logic_table[3] := 0;
stInitData.ModelParameters.Logic_table[4] := 1;
stInitData.ModelParameters.Logic_table[5] := 1;
stInitData.ModelParameters.Logic_table[6] := 0;
stInitData.ModelParameters.Logic_table[7] := 0;
stInitData.ModelParameters.Logic_table[8] := 1;
stInitData.ModelParameters.Logic_table[9] := 0;
stInitData.ModelParameters.Logic_table[10] := 1;
stInitData.ModelParameters.Logic_table[11] := 1;
stInitData.ModelParameters.Logic_table[12] := 0;
stInitData.ModelParameters.Logic_table[13] := 0;
stInitData.ModelParameters.Logic_table[14] := 0;
stInitData.ModelParameters.Logic_table[15] := 0;
stInitData.ModelParameters.Constant_Value_c := 0;
stInitData.ModelParameters.Memory1_X0_m := 0;
stInitData.ModelParameters.Memory_X0_d := 0;
stInitData.ModelParameters.Logic_table_a[0] := 0;
stInitData.ModelParameters.Logic_table_a[1] := 1;
stInitData.ModelParameters.Logic_table_a[2] := 0;
stInitData.ModelParameters.Logic_table_a[3] := 0;
stInitData.ModelParameters.Logic_table_a[4] := 1;
stInitData.ModelParameters.Logic_table_a[5] := 1;
stInitData.ModelParameters.Logic_table_a[6] := 0;
stInitData.ModelParameters.Logic_table_a[7] := 0;
stInitData.ModelParameters.Logic_table_a[8] := 1;
stInitData.ModelParameters.Logic_table_a[9] := 0;
stInitData.ModelParameters.Logic_table_a[10] := 1;
stInitData.ModelParameters.Logic_table_a[11] := 1;
stInitData.ModelParameters.Logic_table_a[12] := 0;
stInitData.ModelParameters.Logic_table_a[13] := 0;
stInitData.ModelParameters.Logic_table_a[14] := 0;
stInitData.ModelParameters.Logic_table_a[15] := 0;
stInitData.ModelParameters.Constant_Value_p := 0;
stInitData.ModelParameters.Memory1_X0_g := 0;
stInitData.ModelParameters.Memory_X0_h := 0;
stInitData.ModelParameters.Logic_table_e[0] := 0;
stInitData.ModelParameters.Logic_table_e[1] := 1;
stInitData.ModelParameters.Logic_table_e[2] := 0;
stInitData.ModelParameters.Logic_table_e[3] := 0;
stInitData.ModelParameters.Logic_table_e[4] := 1;
stInitData.ModelParameters.Logic_table_e[5] := 1;
stInitData.ModelParameters.Logic_table_e[6] := 0;
stInitData.ModelParameters.Logic_table_e[7] := 0;
stInitData.ModelParameters.Logic_table_e[8] := 1;
stInitData.ModelParameters.Logic_table_e[9] := 0;
stInitData.ModelParameters.Logic_table_e[10] := 1;
stInitData.ModelParameters.Logic_table_e[11] := 1;
stInitData.ModelParameters.Logic_table_e[12] := 0;
stInitData.ModelParameters.Logic_table_e[13] := 0;
stInitData.ModelParameters.Logic_table_e[14] := 0;
stInitData.ModelParameters.Logic_table_e[15] := 0;
stInitData.ModelParameters.Constant_Value_b4 := 0;
stInitData.ModelParameters.Memory1_X0_l := 0;
stInitData.ModelParameters.Memory_X0_j := 0;
stInitData.ModelParameters.Logic_table_l[0] := 0;
stInitData.ModelParameters.Logic_table_l[1] := 1;
stInitData.ModelParameters.Logic_table_l[2] := 0;
stInitData.ModelParameters.Logic_table_l[3] := 0;
stInitData.ModelParameters.Logic_table_l[4] := 1;
stInitData.ModelParameters.Logic_table_l[5] := 1;
stInitData.ModelParameters.Logic_table_l[6] := 0;
stInitData.ModelParameters.Logic_table_l[7] := 0;
stInitData.ModelParameters.Logic_table_l[8] := 1;
stInitData.ModelParameters.Logic_table_l[9] := 0;
stInitData.ModelParameters.Logic_table_l[10] := 1;
stInitData.ModelParameters.Logic_table_l[11] := 1;
stInitData.ModelParameters.Logic_table_l[12] := 0;
stInitData.ModelParameters.Logic_table_l[13] := 0;
stInitData.ModelParameters.Logic_table_l[14] := 0;
stInitData.ModelParameters.Logic_table_l[15] := 0;
stInitData.ModelParameters.Constant_Value_a3 := 0;
stInitData.ModelParameters.Memory_X0_hk := 0;
stInitData.ModelParameters.Memory_X0_l := 0;
stInitData.ModelParameters.Memory_X0_p := 0;
stInitData.ModelParameters.Memory_X0_o := 0;
stInitData.ModelParameters.LatchRising_i.Out_Y0 := 0;
stInitData.ModelParameters.LatchRising_a.Out_Y0 := 0;
stInitData.ModelParameters.run_b.x_ref_Y0[0] := 0;
stInitData.ModelParameters.run_b.x_ref_Y0[1] := 0;
stInitData.ModelParameters.run_b.xdot_ref_Y0[0] := 0;
stInitData.ModelParameters.run_b.xdot_ref_Y0[1] := 0;
stInitData.ModelParameters.run_b.xddot_ref_Y0[0] := 0;
stInitData.ModelParameters.run_b.xddot_ref_Y0[1] := 0;
stInitData.ModelParameters.homingactive_g.x_ref_Y0[0] := 0;
stInitData.ModelParameters.homingactive_g.x_ref_Y0[1] := 0;
stInitData.ModelParameters.homingactive_g.xdot_ref_Y0[0] := 0;
stInitData.ModelParameters.homingactive_g.xdot_ref_Y0[1] := 0;
stInitData.ModelParameters.homingactive_g.xddot_ref_Y0[0] := 0;
stInitData.ModelParameters.homingactive_g.xddot_ref_Y0[1] := 0;
stInitData.ModelParameters.homingactive_g.Constant1_Value := 1;
stInitData.ModelParameters.homingactive_g.One_Value := 1;
stInitData.ModelParameters.homingactive_g.RateLimiter_RisingLim := 0.0001;
stInitData.ModelParameters.homingactive_g.RateLimiter_FallingLim := -0.0002;
stInitData.ModelParameters.homingactive_g.RateLimiter_IC := 0;
stInitData.ModelParameters.homingactive_g.Saturation_UpperSat := 1;
stInitData.ModelParameters.homingactive_g.Saturation_LowerSat := 0;
stInitData.ModelParameters.homingactive_g.Gain1_Gain := 6.283185307179586;
stInitData.ModelParameters.homingactive_g.Gain2_Gain := 0.1591549430918953;
stInitData.ModelParameters.homingactive_g.Saturation_UpperSat_b := 1;
stInitData.ModelParameters.homingactive_g.Saturation_LowerSat_p := 0;
stInitData.ModelParameters.homingactive_g.Constant2_Value[0] := 0;
stInitData.ModelParameters.homingactive_g.Constant2_Value[1] := 0;
stInitData.ModelParameters.homingactive_g.Constant4_Value[0] := 0;
stInitData.ModelParameters.homingactive_g.Constant4_Value[1] := 0;
stInitData.ModelParameters.LatchRising_n.Out_Y0 := 0;
stInitData.ModelParameters.LatchRising_gh.Out_Y0 := 0;
stInitData.ModelParameters.run.x_ref_Y0[0] := 0;
stInitData.ModelParameters.run.x_ref_Y0[1] := 0;
stInitData.ModelParameters.run.xdot_ref_Y0[0] := 0;
stInitData.ModelParameters.run.xdot_ref_Y0[1] := 0;
stInitData.ModelParameters.run.xddot_ref_Y0[0] := 0;
stInitData.ModelParameters.run.xddot_ref_Y0[1] := 0;
stInitData.ModelParameters.homingactive.x_ref_Y0[0] := 0;
stInitData.ModelParameters.homingactive.x_ref_Y0[1] := 0;
stInitData.ModelParameters.homingactive.xdot_ref_Y0[0] := 0;
stInitData.ModelParameters.homingactive.xdot_ref_Y0[1] := 0;
stInitData.ModelParameters.homingactive.xddot_ref_Y0[0] := 0;
stInitData.ModelParameters.homingactive.xddot_ref_Y0[1] := 0;
stInitData.ModelParameters.homingactive.Constant1_Value := 1;
stInitData.ModelParameters.homingactive.One_Value := 1;
stInitData.ModelParameters.homingactive.RateLimiter_RisingLim := 0.0001;
stInitData.ModelParameters.homingactive.RateLimiter_FallingLim := -0.0002;
stInitData.ModelParameters.homingactive.RateLimiter_IC := 0;
stInitData.ModelParameters.homingactive.Saturation_UpperSat := 1;
stInitData.ModelParameters.homingactive.Saturation_LowerSat := 0;
stInitData.ModelParameters.homingactive.Gain1_Gain := 6.283185307179586;
stInitData.ModelParameters.homingactive.Gain2_Gain := 0.1591549430918953;
stInitData.ModelParameters.homingactive.Saturation_UpperSat_b := 1;
stInitData.ModelParameters.homingactive.Saturation_LowerSat_p := 0;
stInitData.ModelParameters.homingactive.Constant2_Value[0] := 0;
stInitData.ModelParameters.homingactive.Constant2_Value[1] := 0;
stInitData.ModelParameters.homingactive.Constant4_Value[0] := 0;
stInitData.ModelParameters.homingactive.Constant4_Value[1] := 0;
stInitData.ContextInfoArr_0_TaskOidHdr.indexGroup := 0;
stInitData.ContextInfoArr_0_TaskOidHdr.indexOffset := 16#03002060;
stInitData.ContextInfoArr_0_TaskOidHdr.cbData := SIZEOF(stInitData.ContextInfoArr_0_TaskOid);
stInitData.ContextInfoArr_0_TaskPriorityHdr.indexGroup := 0;
stInitData.ContextInfoArr_0_TaskPriorityHdr.indexOffset := 16#03002070;
stInitData.ContextInfoArr_0_TaskPriorityHdr.cbData := SIZEOF(stInitData.ContextInfoArr_0_TaskPriority);
stInitData.ContextInfoArr_0_TaskCycleTimeNsHdr.indexGroup := 0;
stInitData.ContextInfoArr_0_TaskCycleTimeNsHdr.indexOffset := 16#03002080;
stInitData.ContextInfoArr_0_TaskCycleTimeNsHdr.cbData := SIZEOF(stInitData.ContextInfoArr_0_TaskCycleTimeNs);
stInitData.ContextInfoArr_0_TaskPortHdr.indexGroup := 0;
stInitData.ContextInfoArr_0_TaskPortHdr.indexOffset := 16#03002090;
stInitData.ContextInfoArr_0_TaskPortHdr.cbData := SIZEOF(stInitData.ContextInfoArr_0_TaskPort);
stInitData.ContextInfoArr_0_TaskSortOrderHdr.indexGroup := 0;
stInitData.ContextInfoArr_0_TaskSortOrderHdr.indexOffset := 16#030020b0;
stInitData.ContextInfoArr_0_TaskSortOrderHdr.cbData := SIZEOF(stInitData.ContextInfoArr_0_TaskSortOrder);
stInitData.Header.cbData := SIZEOF(stInitData)-SIZEOF(stInitData.Header);
stInitData.Header.uiElmCnt := 12;


// set pointer to InitData structure
SetInitDataInfo(ADR(stInitData));

// set DataArea information
SetDataAreaInfo(ADR(arrDataAreas),2);
arrDataAreas[1].nDataAreaId := 0;
arrDataAreas[1].nSize := SIZEOF(stInput);
arrDataAreas[1].pPlcVar := ADR(stInput);
arrDataAreas[1].pModuleProcImg := 0;
arrDataAreas[1].eDataAreaType := E_TcMatSimDataAreaType.InputDst;
arrDataAreas[2].nDataAreaId := 1;
arrDataAreas[2].nSize := SIZEOF(stOutput);
arrDataAreas[2].pPlcVar := ADR(stOutput);
arrDataAreas[2].pModuleProcImg := 0;
arrDataAreas[2].eDataAreaType := E_TcMatSimDataAreaType.OutputSrc;


// initialize basic interface pointers and return
FB_init := SUCCEEDED(Init(oid));
                  
                
END_METHOD

METHOD Execute : HRESULT
                  
IF (SUCCEEDED(hResult)) THEN
  hResult := VerifyParameters();
END_IF

	// update DataArea information
SetDataAreaInfo(ADR(arrDataAreas),2);
	
	// call base method
Execute := SUPER^.Execute();
                  
                
END_METHOD

{attribute 'object_name' := 'VerifyParameters'}
METHOD VerifyParameters : HRESULT
  VAR
    moduleCallByParam : TctModuleCallByType;
  END_VAR
                  
IF (bParametersVerified) THEN
  VerifyParameters := Tc2_System.E_HRESULTAdsErr.HRESULT_ADS_NOERROR;
ELSE
  VerifyParameters := GetObjPara(stInitData.CallByHdr.indexOffset,SIZEOF(moduleCallByParam),ADR(moduleCallByParam));
  
  // check the "CallBy" parameter to be set to "Module"
  IF (SUCCEEDED(VerifyParameters) AND (moduleCallByParam <> TctModuleCallByType.Module)) THEN
      VerifyParameters := Tc2_System.E_HRESULTAdsErr.INVALIDPARM;
  END_IF
  
  // set the parameters verified flag
  bParametersVerified := SUCCEEDED(VerifyParameters);
END_IF
                  
                
END_METHOD

PROPERTY InitData : ST_ModelBase2FM_InitData
GET
                    InitData := stInitData;
                  
END_GET
SET
                    stInitData := InitData;
                  
END_SET
END_PROPERTY
END_FUNCTION_BLOCK
